# EPICS autosave request: iocs/andor3IOC/iocBoot/iocAndor3/auto_settings.req
file "andor3_settings.req",       P=$(P),  R=cam1:
file "NDStdArrays_settings.req",  P=$(P),  R=image1:
file "commonPlugin_settings.req", P=$(P)
